DATA_BLOCK "iDB_TRN_Tank_Log_3"
{ S7_Optimized_Access := 'FALSE' }
FAMILY : Archive
VERSION : 1.2
NON_RETAIN
"FB_Tank_Logic"

BEGIN

END_DATA_BLOCK

